FUNCTION_BLOCK ABSTRACT SSC_MoveWorkpiece_Base EXTENDS ControlPrimitiveBase
VAR_INPUT
END_VAR
VAR_OUTPUT
END_VAR
VAR
	m_ptrSSC: POINTER TO SmallSortingConveyor;
	
	m_step: INT := 0;
	m_TurnSwitch : BOOL;
END_VAR

SUPER^();

METHOD  Abort : BOOL
VAR_INPUT
END_VAR
m_ptrSSC^.METH_ConveyorStop();
m_ptrSSC^.METH_Switch_Retract();
Abort := TRUE;
END_METHOD

METHOD PROTECTED ABSTRACT AtTarget : BOOL
VAR_INPUT
END_VAR
END_METHOD

(* Execution logic of this Control Primitive. *)
METHOD PROTECTED ExecuteInternal : BOOL
VAR_INPUT
	i_params: ParameterSet;
END_VAR
CASE m_step OF
	0: // to target	
	IF NOT AtTarget() THEN
		m_ptrSSC^.METH_ConveyorForward();
		IF m_TurnSwitch THEN
			m_ptrSSC^.METH_Switch_Extend();
		END_IF
		m_step := 1;
	END_IF
		
	1:
	IF AtTarget() THEN
		m_ptrSSC^.METH_ConveyorStop();
		IF NOT m_TurnSwitch THEN
			m_ptrSSC^.METH_Switch_Retract();
		END_IF
		m_step := 0;
		ExecuteInternal := TRUE;
	END_IF
		
END_CASE
END_METHOD

END_FUNCTION_BLOCK

(* stored: Version 1.1.0.1, ProductVersion 3.1.4024.12
   POU SSC_MoveWorkpiece_Base: Id {8e09285d-7648-414c-b26c-79d4ab2cbbba}, SpecialFunc None
   Method Abort: Id {20582275-4786-4fc3-aaa7-2a8d5780272b}
   Method AtTarget: Id {393942fe-02f0-426a-93b7-0440a84d3010}
   Method ExecuteInternal: Id {8225cc3c-78ee-48a5-9743-e249f8ff9ad9} *)
